FUNCTION_BLOCK SawmillModule
  (* Standard: 61499-2 *)
  (* Version 0.1, 2017-00-16, hpea485, UOA *)
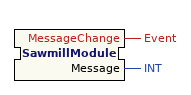
  EVENT_OUTPUT
    MessageChange;
  END_EVENT
  VAR_OUTPUT
    Message : INT;
  END_VAR
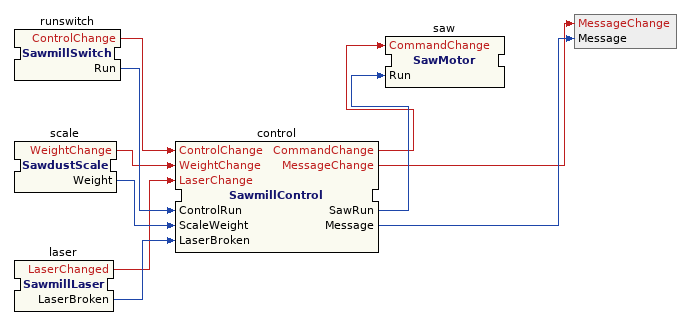
  FBS
    runswitch : SawmillSwitch;
    saw : SawMotor;
    scale : SawdustScale;
    laser : SawmillLaser;
    control : SawmillControl;
  END_FBS
  EVENT_CONNECTIONS
    control.MessageChange TO MessageChange;
    runswitch.ControlChange TO control.ControlChange;
    scale.WeightChange TO control.WeightChange;
    laser.LaserChanged TO control.LaserChange;
    control.CommandChange TO saw.CommandChange;
  END_CONNECTIONS
  DATA_CONNECTIONS
    control.Message TO Message;
    runswitch.Run TO control.ControlRun;
    scale.Weight TO control.ScaleWeight;
    laser.LaserBroken TO control.LaserBroken;
    control.SawRun TO saw.Run;
  END_CONNECTIONS
END_FUNCTION_BLOCK
